LIN {X 0,Y 124.795,Z 460.274,A -85,B 0,C 180,E1 -30071.887,E2 -30071.887} C_VEL
LIN {X 0,Y 121.528,Z 472.694,A -85,B 0,C 180,E1 -30072.738,E2 -30072.738} C_VEL
LIN {X 0,Y 116.919,Z 485.082,A -85,B 0,C 180,E1 -30073.871,E2 -30073.871} C_VEL
LIN {X 0,Y 111.289,Z 496.4,A -85,B 0,C 180,E1 -30075.19,E2 -30075.19} C_VEL
LIN {X 0,Y 104.608,Z 507.03,A -85,B 0,C 180,E1 -30076.792,E2 -30076.792} C_VEL
LIN {X 0,Y 99.806,Z 513.527,A -85,B 0,C 180,E1 -30078.083,E2 -30078.083} C_VEL
LIN {X 0,Y 91.983,Z 522.53,A -85,B 0,C 180,E1 -30080.618,E2 -30080.618} C_VEL
LIN {X 0,Y 85.139,Z 529.183,A -85,B 0,C 180,E1 -30083.105,E2 -30083.105} C_VEL
LIN {X 0,Y 80.808,Z 532.805,A -85,B 0,C 180,E1 -30084.368,E2 -30084.368} C_VEL
LIN {X 0,Y 69.477,Z 540.471,A -85,B 0,C 180,E1 -30086.084,E2 -30086.084} C_VEL
LIN {X 0,Y 62.854,Z 544.286,A -85,B 0,C 180,E1 -30087.829,E2 -30087.829} C_VEL
LIN {X 0,Y 59.746,Z 545.964,A -85,B 0,C 180,E1 -30089.445,E2 -30089.445} C_VEL
LIN {X 0,Y 51.744,Z 549.908,A -85,B 0,C 180,E1 -30095.42,E2 -30095.42} C_VEL
LIN {X 0,Y 46.39,Z 552.162,A -85,B 0,C 180,E1 -30100.758,E2 -30100.758} C_VEL
LIN {X 0,Y 41.567,Z 553.982,A -85,B 0,C 180,E1 -30107.445,E2 -30107.445} C_VEL
LIN {X 0,Y 37.649,Z 555.304,A -85,B 0,C 180,E1 -30115.945,E2 -30115.945} C_VEL
LIN {X 0,Y 32.48,Z 556.841,A -85,B 0,C 180,E1 -30137.504,E2 -30137.504} C_VEL
LIN {X 0,Y 31.773,Z 557.059,A -85,B 0,C 180,E1 -30150,E2 -30150} C_VEL
LIN {X 0,Y 32.479,Z 556.865,A -85,B 0,C 180,E1 -30162.497,E2 -30162.497} C_VEL
LIN {X 0,Y 37.641,Z 555.359,A -85,B 0,C 180,E1 -30184.064,E2 -30184.064} C_VEL
LIN {X 0,Y 41.551,Z 554.064,A -85,B 0,C 180,E1 -30192.575,E2 -30192.575} C_VEL
LIN {X 0,Y 49.098,Z 551.206,A -85,B 0,C 180,E1 -30201.931,E2 -30201.931} C_VEL
LIN {X 0,Y 57.415,Z 547.366,A -85,B 0,C 180,E1 -30208.962,E2 -30208.962} C_VEL
LIN {X 0,Y 66.482,Z 542.269,A -85,B 0,C 180,E1 -30214.662,E2 -30214.662} C_VEL
LIN {X 0,Y 77.008,Z 535.01,A -85,B 0,C 180,E1 -30219.299,E2 -30219.299} C_VEL
LIN {X 0,Y 86.535,Z 526.968,A -85,B 0,C 180,E1 -30222.606,E2 -30222.606} C_VEL
LIN {X 0,Y 94.587,Z 518.728,A -85,B 0,C 180,E1 -30224.997,E2 -30224.997} C_VEL
LIN {X 0,Y 101.933,Z 509.667,A -85,B 0,C 180,E1 -30226.871,E2 -30226.871} C_VEL
LIN {X 0,Y 109.586,Z 498.077,A -85,B 0,C 180,E1 -30228.344,E2 -30228.344} C_VEL
LIN {X 0,Y 115.483,Z 486.708,A -85,B 0,C 180,E1 -30229.556,E2 -30229.556} C_VEL
LIN {X 0,Y 120.111,Z 475.001,A -85,B 0,C 180,E1 -30230.442,E2 -30230.442} C_VEL
LIN {X 0,Y 122.962,Z 465.192,A -85,B 0,C 180,E1 -30231.247,E2 -30231.247} C_VEL
LIN {X 0,Y 122.843,Z 462.958,A -85,B 0,C 180,E1 -30234.665,E2 -30234.665} C_VEL
LIN {X 0,Y 122.946,Z 461.545,A -85,B 0,C 180,E1 -30238.362,E2 -30238.362} C_VEL
LIN {X 0,Y 122.98,Z 461.9,A -85,B 0,C 180,E1 -30240.818,E2 -30240.818} C_VEL
LIN {X 0,Y 123.076,Z 463.09,A -85,B 0,C 180,E1 -30243.273,E2 -30243.273} C_VEL
LIN {X 0,Y 122.853,Z 466.21,A -85,B 0,C 180,E1 -30245.468,E2 -30245.468} C_VEL
LIN {X 0,Y 120.841,Z 474.449,A -85,B 0,C 180,E1 -30246.208,E2 -30246.208} C_VEL
LIN {X 0,Y 116.49,Z 486.717,A -85,B 0,C 180,E1 -30246.694,E2 -30246.694} C_VEL
LIN {X 0,Y 110.404,Z 499.391,A -85,B 0,C 180,E1 -30247.354,E2 -30247.354} C_VEL
LIN {X 0,Y 103.852,Z 510.17,A -85,B 0,C 180,E1 -30248.229,E2 -30248.229} C_VEL
LIN {X 0,Y 96.119,Z 520.374,A -85,B 0,C 180,E1 -30249.225,E2 -30249.225} C_VEL
LIN {X 0,Y 87.628,Z 529.627,A -85,B 0,C 180,E1 -30250.746,E2 -30250.746} C_VEL
LIN {X 0,Y 77.518,Z 538.659,A -85,B 0,C 180,E1 -30252.94,E2 -30252.94} C_VEL
LIN {X 0,Y 67.63,Z 545.987,A -85,B 0,C 180,E1 -30256.007,E2 -30256.007} C_VEL
LIN {X 0,Y 56.495,Z 552.728,A -85,B 0,C 180,E1 -30261.095,E2 -30261.095} C_VEL
LIN {X 0,Y 47.545,Z 557.256,A -85,B 0,C 180,E1 -30267.515,E2 -30267.515} C_VEL
LIN {X 0,Y 39.516,Z 560.732,A -85,B 0,C 180,E1 -30276.84,E2 -30276.84} C_VEL
LIN {X 0,Y 33.166,Z 563.257,A -85,B 0,C 180,E1 -30290.527,E2 -30290.527} C_VEL
LIN {X 0,Y 29.149,Z 565.212,A -85,B 0,C 180,E1 -30316.048,E2 -30316.048} C_VEL
LIN {X 0,Y 29.564,Z 565.594,A -85,B 0,C 180,E1 -30330,E2 -30330} C_VEL
LIN {X 0,Y 29.186,Z 565.111,A -85,B 0,C 180,E1 -30345.59,E2 -30345.59} C_VEL
LIN {X 0,Y 33.151,Z 563.208,A -85,B 0,C 180,E1 -30369.493,E2 -30369.493} C_VEL
LIN {X 0,Y 39.516,Z 560.656,A -85,B 0,C 180,E1 -30383.159,E2 -30383.159} C_VEL
LIN {X 0,Y 47.544,Z 557.144,A -85,B 0,C 180,E1 -30392.486,E2 -30392.486} C_VEL
LIN {X 0,Y 56.494,Z 552.58,A -85,B 0,C 180,E1 -30398.907,E2 -30398.907} C_VEL
LIN {X 0,Y 65.996,Z 546.848,A -85,B 0,C 180,E1 -30403.416,E2 -30403.416} C_VEL
LIN {X 0,Y 75.851,Z 539.771,A -85,B 0,C 180,E1 -30406.622,E2 -30406.622} C_VEL
LIN {X 0,Y 85.935,Z 530.978,A -85,B 0,C 180,E1 -30408.925,E2 -30408.925} C_VEL
LIN {X 0,Y 94.423,Z 521.995,A -85,B 0,C 180,E1 -30410.468,E2 -30410.468} C_VEL
LIN {X 0,Y 102.994,Z 510.982,A -85,B 0,C 180,E1 -30411.657,E2 -30411.657} C_VEL
LIN {X 0,Y 110.23,Z 499.134,A -85,B 0,C 180,E1 -30412.611,E2 -30412.611} C_VEL
LIN {X 0,Y 116.308,Z 486.38,A -85,B 0,C 180,E1 -30413.295,E2 -30413.295} C_VEL
LIN {X 0,Y 120.833,Z 473.286,A -85,B 0,C 180,E1 -30413.82,E2 -30413.82} C_VEL
LIN {X 0,Y 122.61,Z 465.716,A -85,B 0,C 180,E1 -30414.621,E2 -30414.621} C_VEL
LIN {X 0,Y 122.799,Z 462.414,A -85,B 0,C 180,E1 -30417.13,E2 -30417.13} C_VEL
LIN {X 0,Y 122.712,Z 461.196,A -85,B 0,C 180,E1 -30420,E2 -30420} C_VEL
LIN {X 0,Y 122.655,Z 461.282,A -85,B 0,C 180,E1 -30422.052,E2 -30422.052} C_VEL
LIN {X 0,Y 122.586,Z 463.339,A -85,B 0,C 180,E1 -30426.584,E2 -30426.584} C_VEL
LIN {X 0,Y 122.689,Z 464.933,A -85,B 0,C 180,E1 -30428.843,E2 -30428.843} C_VEL
LIN {X 0,Y 118.804,Z 477.683,A -85,B 0,C 180,E1 -30429.782,E2 -30429.782} C_VEL
LIN {X 0,Y 113.601,Z 489.945,A -85,B 0,C 180,E1 -30430.842,E2 -30430.842} C_VEL
LIN {X 0,Y 107.762,Z 500.568,A -85,B 0,C 180,E1 -30431.972,E2 -30431.972} C_VEL
LIN {X 0,Y 101.946,Z 509.183,A -85,B 0,C 180,E1 -30433.161,E2 -30433.161} C_VEL
LIN {X 0,Y 94.591,Z 518.343,A -85,B 0,C 180,E1 -30435.014,E2 -30435.014} C_VEL
LIN {X 0,Y 86.541,Z 526.664,A -85,B 0,C 180,E1 -30437.407,E2 -30437.407} C_VEL
LIN {X 0,Y 77.004,Z 534.762,A -85,B 0,C 180,E1 -30440.694,E2 -30440.694} C_VEL
LIN {X 0,Y 66.818,Z 541.857,A -85,B 0,C 180,E1 -30445.202,E2 -30445.202} C_VEL
LIN {X 0,Y 59.746,Z 545.964,A -85,B 0,C 180,E1 -30449.445,E2 -30449.445} C_VEL
LIN {X 0,Y 54.965,Z 548.348,A -85,B 0,C 180,E1 -30451.99,E2 -30451.99} C_VEL
LIN {X 0,Y 46.173,Z 551.895,A -85,B 0,C 180,E1 -30455.343,E2 -30455.343} C_VEL
LIN {X 0,Y 37.449,Z 554.767,A -85,B 0,C 180,E1 -30460.448,E2 -30460.448} C_VEL
LIN {X 0,Y 33.098,Z 555.966,A -85,B 0,C 180,E1 -30466.541,E2 -30466.541} C_VEL
LIN {X 0,Y 28.156,Z 557.247,A -85,B 0,C 180,E1 -30480.053,E2 -30480.053} C_VEL
LIN {X 0,Y 25.663,Z 557.819,A -85,B 0,C 180,E1 -30494.107,E2 -30494.107} C_VEL
LIN {X 0,Y 24.745,Z 558.037,A -85,B 0,C 180,E1 -30510,E2 -30510} C_VEL
LIN {X 0,Y 25.663,Z 557.843,A -85,B 0,C 180,E1 -30525.894,E2 -30525.894} C_VEL
LIN {X 0,Y 32.06,Z 556.337,A -85,B 0,C 180,E1 -30551.119,E2 -30551.119} C_VEL
LIN {X 0,Y 36.682,Z 555.042,A -85,B 0,C 180,E1 -30560.027,E2 -30560.027} C_VEL
LIN {X 0,Y 45.105,Z 552.183,A -85,B 0,C 180,E1 -30568.977,E2 -30568.977} C_VEL
LIN {X 0,Y 54.128,Z 548.343,A -85,B 0,C 180,E1 -30575.35,E2 -30575.35} C_VEL
LIN {X 0,Y 63.791,Z 543.246,A -85,B 0,C 180,E1 -30580.377,E2 -30580.377} C_VEL
LIN {X 0,Y 74.813,Z 535.986,A -85,B 0,C 180,E1 -30584.341,E2 -30584.341} C_VEL
LIN {X 0,Y 84.699,Z 527.944,A -85,B 0,C 180,E1 -30587.148,E2 -30587.148} C_VEL
LIN {X 0,Y 93.015,Z 519.704,A -85,B 0,C 180,E1 -30589.184,E2 -30589.184} C_VEL
LIN {X 0,Y 100.571,Z 510.641,A -85,B 0,C 180,E1 -30590.77,E2 -30590.77} C_VEL
LIN {X 0,Y 108.381,Z 499.057,A -85,B 0,C 180,E1 -30591.985,E2 -30591.985} C_VEL
LIN {X 0,Y 114.078,Z 488.375,A -85,B 0,C 180,E1 -30592.973,E2 -30592.973} C_VEL
LIN {X 0,Y 118.98,Z 476.468,A -85,B 0,C 180,E1 -30593.757,E2 -30593.757} C_VEL
LIN {X 0,Y 120.929,Z 470.35,A -85,B 0,C 180,E1 -30594.202,E2 -30594.202} C_VEL
LIN {X 0,Y 121.098,Z 468.993,A -85,B 0,C 180,E1 -30597.089,E2 -30597.089} C_VEL
LIN {X 0,Y 121.221,Z 468.565,A -85,B 0,C 180,E1 -30598.339,E2 -30598.339} C_VEL
LIN {X 0,Y 121.3,Z 468.744,A -85,B 0,C 180,E1 -30600.456,E2 -30600.456} C_VEL
LIN {X 0,Y 121.262,Z 469.63,A -85,B 0,C 180,E1 -30602.107,E2 -30602.107} C_VEL
LIN {X 0,Y 121.188,Z 470.103,A -85,B 0,C 180,E1 -30602.483,E2 -30602.483} C_VEL
LIN {X 0,Y 119.624,Z 475.528,A -85,B 0,C 180,E1 -30602.868,E2 -30602.868} C_VEL
LIN {X 0,Y 114.846,Z 488.092,A -85,B 0,C 180,E1 -30603.275,E2 -30603.275} C_VEL
LIN {X 0,Y 108.868,Z 499.965,A -85,B 0,C 180,E1 -30603.741,E2 -30603.741} C_VEL
LIN {X 0,Y 102.205,Z 510.441,A -85,B 0,C 180,E1 -30604.394,E2 -30604.394} C_VEL
LIN {X 0,Y 93.504,Z 521.362,A -85,B 0,C 180,E1 -30605.198,E2 -30605.198} C_VEL
LIN {X 0,Y 84.856,Z 530.29,A -85,B 0,C 180,E1 -30606.355,E2 -30606.355} C_VEL
LIN {X 0,Y 74.525,Z 539.006,A -85,B 0,C 180,E1 -30608.038,E2 -30608.038} C_VEL
LIN {X 0,Y 64.33,Z 546.043,A -85,B 0,C 180,E1 -30610.508,E2 -30610.508} C_VEL
LIN {X 0,Y 54.331,Z 551.733,A -85,B 0,C 180,E1 -30614.035,E2 -30614.035} C_VEL
LIN {X 0,Y 44.697,Z 556.263,A -85,B 0,C 180,E1 -30619.367,E2 -30619.367} C_VEL
LIN {X 0,Y 35.683,Z 559.735,A -85,B 0,C 180,E1 -30627.59,E2 -30627.59} C_VEL
LIN {X 0,Y 28.005,Z 562.26,A -85,B 0,C 180,E1 -30641.163,E2 -30641.163} C_VEL
LIN {X 0,Y 22.262,Z 564.215,A -85,B 0,C 180,E1 -30671.597,E2 -30671.597} C_VEL
LIN {X 0,Y 22.418,Z 564.6,A -85,B 0,C 180,E1 -30690,E2 -30690} C_VEL
LIN {X 0,Y 24.248,Z 563.393,A -85,B 0,C 180,E1 -30725.427,E2 -30725.427} C_VEL
LIN {X 0,Y 32.913,Z 560.629,A -85,B 0,C 180,E1 -30748.663,E2 -30748.663} C_VEL
LIN {X 0,Y 41.593,Z 557.452,A -85,B 0,C 180,E1 -30758.33,E2 -30758.33} C_VEL
LIN {X 0,Y 51.072,Z 553.254,A -85,B 0,C 180,E1 -30764.419,E2 -30764.419} C_VEL
LIN {X 0,Y 62.643,Z 546.894,A -85,B 0,C 180,E1 -30769.008,E2 -30769.008} C_VEL
LIN {X 0,Y 72.817,Z 540.04,A -85,B 0,C 180,E1 -30771.596,E2 -30771.596} C_VEL
LIN {X 0,Y 83.132,Z 531.612,A -85,B 0,C 180,E1 -30773.378,E2 -30773.378} C_VEL
LIN {X 0,Y 91.778,Z 522.981,A -85,B 0,C 180,E1 -30774.543,E2 -30774.543} C_VEL
LIN {X 0,Y 99.596,Z 513.552,A -85,B 0,C 180,E1 -30775.353,E2 -30775.353} C_VEL
LIN {X 0,Y 106.763,Z 502.925,A -85,B 0,C 180,E1 -30776.103,E2 -30776.103} C_VEL
LIN {X 0,Y 113.161,Z 491.081,A -85,B 0,C 180,E1 -30776.6,E2 -30776.6} C_VEL
LIN {X 0,Y 118.133,Z 478.999,A -85,B 0,C 180,E1 -30776.993,E2 -30776.993} C_VEL
LIN {X 0,Y 120.408,Z 471.722,A -85,B 0,C 180,E1 -30777.355,E2 -30777.355} C_VEL
LIN {X 0,Y 120.958,Z 469.658,A -85,B 0,C 180,E1 -30777.615,E2 -30777.615} C_VEL
LIN {X 0,Y 121.06,Z 468.907,A -85,B 0,C 180,E1 -30778.335,E2 -30778.335} C_VEL
LIN {X 0,Y 121.05,Z 468.267,A -85,B 0,C 180,E1 -30780,E2 -30780} C_VEL
LIN {X 0,Y 120.933,Z 468.333,A -85,B 0,C 180,E1 -30782.082,E2 -30782.082} C_VEL
LIN {X 0,Y 120.685,Z 469.949,A -85,B 0,C 180,E1 -30785.763,E2 -30785.763} C_VEL
LIN {X 0,Y 116.757,Z 481.449,A -85,B 0,C 180,E1 -30786.623,E2 -30786.623} C_VEL
LIN {X 0,Y 111.443,Z 493.006,A -85,B 0,C 180,E1 -30787.52,E2 -30787.52} C_VEL
LIN {X 0,Y 104.833,Z 504.139,A -85,B 0,C 180,E1 -30788.575,E2 -30788.575} C_VEL
LIN {X 0,Y 98.047,Z 513.408,A -85,B 0,C 180,E1 -30789.742,E2 -30789.742} C_VEL
LIN {X 0,Y 89.683,Z 522.835,A -85,B 0,C 180,E1 -30791.609,E2 -30791.609} C_VEL
LIN {X 0,Y 81.375,Z 530.559,A -85,B 0,C 180,E1 -30793.69,E2 -30793.69} C_VEL
LIN {X 0,Y 71.381,Z 538.2,A -85,B 0,C 180,E1 -30796.769,E2 -30796.769} C_VEL
LIN {X 0,Y 60.343,Z 544.993,A -85,B 0,C 180,E1 -30801.296,E2 -30801.296} C_VEL
LIN {X 0,Y 51.049,Z 549.593,A -85,B 0,C 180,E1 -30806.511,E2 -30806.511} C_VEL
LIN {X 0,Y 42.137,Z 553.142,A -85,B 0,C 180,E1 -30813.496,E2 -30813.496} C_VEL
LIN {X 0,Y 36.696,Z 554.961,A -85,B 0,C 180,E1 -30819.999,E2 -30819.999} C_VEL
LIN {X 0,Y 33.098,Z 555.966,A -85,B 0,C 180,E1 -30826.541,E2 -30826.541} C_VEL
LIN {X 0,Y 29.203,Z 557.017,A -85,B 0,C 180,E1 -30834.481,E2 -30834.481} C_VEL
LIN {X 0,Y 22.567,Z 558.393,A -85,B 0,C 180,E1 -30850.678,E2 -30850.678} C_VEL
LIN {X 0,Y 18.927,Z 558.932,A -85,B 0,C 180,E1 -30870.447,E2 -30870.447} C_VEL
LIN {X 0,Y 18.751,Z 558.874,A -85,B 0,C 180,E1 -30888.621,E2 -30888.621} C_VEL
LIN {X 0,Y 19.331,Z 558.747,A -85,B 0,C 180,E1 -30894.322,E2 -30894.322} C_VEL
LIN {X 0,Y 27.16,Z 557.315,A -85,B 0,C 180,E1 -30920.92,E2 -30920.92} C_VEL
LIN {X 0,Y 32.613,Z 556.019,A -85,B 0,C 180,E1 -30929.538,E2 -30929.538} C_VEL
LIN {X 0,Y 41.918,Z 553.16,A -85,B 0,C 180,E1 -30937.238,E2 -30937.238} C_VEL
LIN {X 0,Y 51.593,Z 549.319,A -85,B 0,C 180,E1 -30942.462,E2 -30942.462} C_VEL
LIN {X 0,Y 61.786,Z 544.222,A -85,B 0,C 180,E1 -30946.527,E2 -30946.527} C_VEL
LIN {X 0,Y 73.229,Z 536.962,A -85,B 0,C 180,E1 -30949.643,E2 -30949.643} C_VEL
LIN {X 0,Y 83.418,Z 528.919,A -85,B 0,C 180,E1 -30951.86,E2 -30951.86} C_VEL
LIN {X 0,Y 91.955,Z 520.679,A -85,B 0,C 180,E1 -30953.491,E2 -30953.491} C_VEL
LIN {X 0,Y 99.684,Z 511.616,A -85,B 0,C 180,E1 -30954.767,E2 -30954.767} C_VEL
LIN {X 0,Y 107.626,Z 500.031,A -85,B 0,C 180,E1 -30955.693,E2 -30955.693} C_VEL
LIN {X 0,Y 114.008,Z 488.167,A -85,B 0,C 180,E1 -30956.571,E2 -30956.571} C_VEL
LIN {X 0,Y 118.621,Z 476.847,A -85,B 0,C 180,E1 -30957.16,E2 -30957.16} C_VEL
LIN {X 0,Y 118.992,Z 475.748,A -85,B 0,C 180,E1 -30957.421,E2 -30957.421} C_VEL
LIN {X 0,Y 119.18,Z 475.36,A -85,B 0,C 180,E1 -30959.117,E2 -30959.117} C_VEL
LIN {X 0,Y 118.829,Z 476.478,A -85,B 0,C 180,E1 -30959.489,E2 -30959.489} C_VEL
LIN {X 0,Y 114.05,Z 488.497,A -85,B 0,C 180,E1 -30959.755,E2 -30959.755} C_VEL
LIN {X 0,Y 107.61,Z 500.694,A -85,B 0,C 180,E1 -30960.04,E2 -30960.04} C_VEL
LIN {X 0,Y 100.151,Z 511.824,A -85,B 0,C 180,E1 -30960.499,E2 -30960.499} C_VEL
LIN {X 0,Y 91.375,Z 522.339,A -85,B 0,C 180,E1 -30960.965,E2 -30960.965} C_VEL
LIN {X 0,Y 82.614,Z 530.899,A -85,B 0,C 180,E1 -30961.699,E2 -30961.699} C_VEL
LIN {X 0,Y 72.12,Z 539.275,A -85,B 0,C 180,E1 -30962.774,E2 -30962.774} C_VEL
LIN {X 0,Y 61.683,Z 546.092,A -85,B 0,C 180,E1 -30964.492,E2 -30964.492} C_VEL
LIN {X 0,Y 49.633,Z 552.395,A -85,B 0,C 180,E1 -30967.615,E2 -30967.615} C_VEL
LIN {X 0,Y 39.514,Z 556.555,A -85,B 0,C 180,E1 -30971.978,E2 -30971.978} C_VEL
LIN {X 0,Y 29.821,Z 559.703,A -85,B 0,C 180,E1 -30979.492,E2 -30979.492} C_VEL
LIN {X 0,Y 18.878,Z 562.432,A -85,B 0,C 180,E1 -31001.878,E2 -31001.878} C_VEL
LIN {X 0,Y 15.512,Z 563.264,A -85,B 0,C 180,E1 -31024.972,E2 -31024.972} C_VEL
LIN {X 0,Y 15.27,Z 563.605,A -85,B 0,C 180,E1 -31050,E2 -31050} C_VEL
LIN {X 0,Y 15.625,Z 563.196,A -85,B 0,C 180,E1 -31076.729,E2 -31076.729} C_VEL
LIN {X 0,Y 23.896,Z 561.212,A -85,B 0,C 180,E1 -31111.921,E2 -31111.921} C_VEL
LIN {X 0,Y 32.985,Z 558.661,A -85,B 0,C 180,E1 -31123.491,E2 -31123.491} C_VEL
LIN {X 0,Y 42.859,Z 555.153,A -85,B 0,C 180,E1 -31129.69,E2 -31129.69} C_VEL
LIN {X 0,Y 53.052,Z 550.587,A -85,B 0,C 180,E1 -31133.482,E2 -31133.482} C_VEL
LIN {X 0,Y 63.418,Z 544.864,A -85,B 0,C 180,E1 -31135.835,E2 -31135.835} C_VEL
LIN {X 0,Y 73.867,Z 537.785,A -85,B 0,C 180,E1 -31137.433,E2 -31137.433} C_VEL
LIN {X 0,Y 84.365,Z 528.994,A -85,B 0,C 180,E1 -31138.447,E2 -31138.447} C_VEL
LIN {X 0,Y 93.13,Z 520.008,A -85,B 0,C 180,E1 -31139.14,E2 -31139.14} C_VEL
LIN {X 0,Y 101.028,Z 510.186,A -85,B 0,C 180,E1 -31139.562,E2 -31139.562} C_VEL
LIN {X 0,Y 107.997,Z 499.508,A -85,B 0,C 180,E1 -31139.977,E2 -31139.977} C_VEL
LIN {X 0,Y 113.917,Z 488.027,A -85,B 0,C 180,E1 -31140.232,E2 -31140.232} C_VEL
LIN {X 0,Y 118.463,Z 476.548,A -85,B 0,C 180,E1 -31140.47,E2 -31140.47} C_VEL
LIN {X 0,Y 118.966,Z 475.014,A -85,B 0,C 180,E1 -31140.666,E2 -31140.666} C_VEL
LIN {X 0,Y 118.737,Z 475.468,A -85,B 0,C 180,E1 -31142.588,E2 -31142.588} C_VEL
LIN {X 0,Y 118.46,Z 476.289,A -85,B 0,C 180,E1 -31142.807,E2 -31142.807} C_VEL
LIN {X 0,Y 114.122,Z 487.13,A -85,B 0,C 180,E1 -31143.45,E2 -31143.45} C_VEL
LIN {X 0,Y 108.358,Z 498.273,A -85,B 0,C 180,E1 -31144.239,E2 -31144.239} C_VEL
LIN {X 0,Y 102.29,Z 507.654,A -85,B 0,C 180,E1 -31144.978,E2 -31144.978} C_VEL
LIN {X 0,Y 96.249,Z 515.433,A -85,B 0,C 180,E1 -31145.809,E2 -31145.809} C_VEL
LIN {X 0,Y 88.537,Z 523.816,A -85,B 0,C 180,E1 -31147.149,E2 -31147.149} C_VEL
LIN {X 0,Y 80.004,Z 531.539,A -85,B 0,C 180,E1 -31148.793,E2 -31148.793} C_VEL
LIN {X 0,Y 69.679,Z 539.18,A -85,B 0,C 180,E1 -31151.227,E2 -31151.227} C_VEL
LIN {X 0,Y 58.161,Z 545.972,A -85,B 0,C 180,E1 -31154.832,E2 -31154.832} C_VEL
LIN {X 0,Y 48.323,Z 550.572,A -85,B 0,C 180,E1 -31159.033,E2 -31159.033} C_VEL
LIN {X 0,Y 38.704,Z 554.121,A -85,B 0,C 180,E1 -31164.783,E2 -31164.783} C_VEL
LIN {X 0,Y 32.624,Z 555.94,A -85,B 0,C 180,E1 -31170.495,E2 -31170.495} C_VEL
LIN {X 0,Y 27.167,Z 557.261,A -85,B 0,C 180,E1 -31179.098,E2 -31179.098} C_VEL
LIN {X 0,Y 19.001,Z 558.797,A -85,B 0,C 180,E1 -31208.293,E2 -31208.293} C_VEL
LIN {X 0,Y 17.717,Z 559.015,A -85,B 0,C 180,E1 -31230,E2 -31230} C_VEL
LIN {X 0,Y 19.331,Z 558.747,A -85,B 0,C 180,E1 -31254.322,E2 -31254.322} C_VEL
LIN {X 0,Y 21.622,Z 558.407,A -85,B 0,C 180,E1 -31269.604,E2 -31269.604} C_VEL
LIN {X 0,Y 26.591,Z 557.523,A -85,B 0,C 180,E1 -31290.188,E2 -31290.188} C_VEL
LIN {X 0,Y 32.138,Z 556.298,A -85,B 0,C 180,E1 -31301.04,E2 -31301.04} C_VEL
LIN {X 0,Y 37.169,Z 554.94,A -85,B 0,C 180,E1 -31305.557,E2 -31305.557} C_VEL
LIN {X 0,Y 38.973,Z 554.373,A -85,B 0,C 180,E1 -31306.367,E2 -31306.367} C_VEL
LIN {X 0,Y 49.927,Z 550.296,A -85,B 0,C 180,E1 -31310.175,E2 -31310.175} C_VEL
LIN {X 0,Y 60.536,Z 545.199,A -85,B 0,C 180,E1 -31313.01,E2 -31313.01} C_VEL
LIN {X 0,Y 72.297,Z 537.938,A -85,B 0,C 180,E1 -31315.13,E2 -31315.13} C_VEL
LIN {X 0,Y 77.5,Z 534.136,A -85,B 0,C 180,E1 -31315.954,E2 -31315.954} C_VEL
LIN {X 0,Y 77.42,Z 534.314,A -85,B 0,C 180,E1 -31316.904,E2 -31316.904} C_VEL
LIN {X 0,Y 66.831,Z 541.875,A -85,B 0,C 180,E1 -31317.455,E2 -31317.455} C_VEL
LIN {X 0,Y 56.245,Z 548,A -85,B 0,C 180,E1 -31318.388,E2 -31318.388} C_VEL
LIN {X 0,Y 45.382,Z 553.025,A -85,B 0,C 180,E1 -31320,E2 -31320} C_VEL
LIN {X 0,Y 35.178,Z 556.708,A -85,B 0,C 180,E1 -31322.684,E2 -31322.684} C_VEL
LIN {X 0,Y 28.249,Z 558.706,A -85,B 0,C 180,E1 -31325.661,E2 -31325.661} C_VEL
LIN {X 0,Y 15.069,Z 561.435,A -85,B 0,C 180,E1 -31341.13,E2 -31341.13} C_VEL
LIN {X 0,Y 9.089,Z 562.332,A -85,B 0,C 180,E1 -31370.642,E2 -31370.642} C_VEL
LIN {X 0,Y 8.13,Z 562.611,A -85,B 0,C 180,E1 -31409.999,E2 -31409.999} C_VEL
LIN {X 0,Y 9.773,Z 562.199,A -85,B 0,C 180,E1 -31455.982,E2 -31455.982} C_VEL
LIN {X 0,Y 21.471,Z 560.212,A -85,B 0,C 180,E1 -31489.092,E2 -31489.092} C_VEL
LIN {X 0,Y 31.704,Z 557.666,A -85,B 0,C 180,E1 -31495.973,E2 -31495.973} C_VEL
LIN {X 0,Y 42.17,Z 554.159,A -85,B 0,C 180,E1 -31499.281,E2 -31499.281} C_VEL
LIN {X 0,Y 52.721,Z 549.592,A -85,B 0,C 180,E1 -31501.212,E2 -31501.212} C_VEL
LIN {X 0,Y 64.887,Z 542.923,A -85,B 0,C 180,E1 -31502.396,E2 -31502.396} C_VEL
LIN {X 0,Y 75.656,Z 535.43,A -85,B 0,C 180,E1 -31503.04,E2 -31503.04} C_VEL
LIN {X 0,Y 77.419,Z 534.054,A -85,B 0,C 180,E1 -31503.095,E2 -31503.095} C_VEL
LIN {X 0,Y 77.496,Z 533.88,A -85,B 0,C 180,E1 -31504.013,E2 -31504.013} C_VEL
LIN {X 0,Y 67.104,Z 541.135,A -85,B 0,C 180,E1 -31505.767,E2 -31505.767} C_VEL
LIN {X 0,Y 56.77,Z 546.952,A -85,B 0,C 180,E1 -31507.958,E2 -31507.958} C_VEL
LIN {X 0,Y 46.508,Z 551.551,A -85,B 0,C 180,E1 -31510.82,E2 -31510.82} C_VEL
LIN {X 0,Y 36.322,Z 555.1,A -85,B 0,C 180,E1 -31514.66,E2 -31514.66} C_VEL
LIN {X 0,Y 29.681,Z 556.92,A -85,B 0,C 180,E1 -31518.716,E2 -31518.716} C_VEL
LIN {X 0,Y 23.379,Z 558.24,A -85,B 0,C 180,E1 -31525.603,E2 -31525.603} C_VEL
LIN {X 0,Y 12.74,Z 559.775,A -85,B 0,C 180,E1 -31556.52,E2 -31556.52} C_VEL
LIN {X 0,Y 10.689,Z 559.993,A -85,B 0,C 180,E1 -31590,E2 -31590} C_VEL
LIN {X 0,Y 13.129,Z 559.741,A -85,B 0,C 180,E1 -31626.192,E2 -31626.192} C_VEL
LIN {X 0,Y 23.375,Z 558.293,A -85,B 0,C 180,E1 -31654.421,E2 -31654.421} C_VEL
LIN {X 0,Y 29.674,Z 556.997,A -85,B 0,C 180,E1 -31661.324,E2 -31661.324} C_VEL
LIN {X 0,Y 38.973,Z 554.373,A -85,B 0,C 180,E1 -31666.367,E2 -31666.367} C_VEL
LIN {X 0,Y 37.594,Z 554.867,A -85,B 0,C 180,E1 -31667.268,E2 -31667.268} C_VEL
LIN {X 0,Y 30.022,Z 557.131,A -85,B 0,C 180,E1 -31667.71,E2 -31667.71} C_VEL
LIN {X 0,Y 17.103,Z 559.779,A -85,B 0,C 180,E1 -31664.889,E2 -31664.889} C_VEL
LIN {X 0,Y 7.659,Z 560.787,A -85,B 0,C 180,E1 -31651.379,E2 -31651.379} C_VEL
LIN {X 0,Y 4.998,Z 560.876,A -85,B 0,C 180,E1 -31633.424,E2 -31633.424} C_VEL
LIN {X 0,Y 7.895,Z 560.753,A -85,B 0,C 180,E1 -31527.109,E2 -31527.109} C_VEL
LIN {X 0,Y 14.44,Z 560.182,A -85,B 0,C 180,E1 -31513.256,E2 -31513.256} C_VEL
LIN {X 0,Y 14.165,Z 560.398,A -85,B 0,C 180,E1 -31507.127,E2 -31507.127} C_VEL
LIN {X 0,Y 0.988,Z 561.618,A -85,B 0,C 180,E1 -31409.995,E2 -31409.995} C_VEL
LIN {X 0,Y 14.164,Z 560.436,A -85,B 0,C 180,E1 -31312.903,E2 -31312.903} C_VEL
LIN {X 0,Y 14.44,Z 560.219,A -85,B 0,C 180,E1 -31306.755,E2 -31306.755} C_VEL
LIN {X 0,Y 4.998,Z 560.876,A -85,B 0,C 180,E1 -31273.424,E2 -31273.424} C_VEL
LIN {X 0,Y 3.94,Z 562.875,A -85,B 0,C 180,E1 -31252.23,E2 -31252.23} C_VEL
LIN {X 0,Y 3.94,Z 600,A -85,B 0,C 180,E1 -31252.23,E2 -31252.23} C_VEL
LIN {X 0,Y 3.94,Z 600,A -85,B 0,C 180,E1 -31252.23,E2 -31252.23}

QRS_NEXT_CUT()

QRS_NEXT()
QRS_HOME()

END
